// TIA Portal V16 export
// export: Created 2024-09-05T17:39:16.5674973Z, ExportSetting WithDefaults, DisplayName Totally Integrated Automation Portal, DisplayVersion V16 Update 6, DisplayName TIA Portal Version Control Interface, DisplayVersion V16 Update 2, DisplayName TIA Portal Openness, DisplayVersion V16 Update 6, DisplayName STEP 7 Professional, DisplayVersion V16 Update 6, DisplayName STEP 7 Safety, DisplayVersion V16, DisplayName WinCC Advanced, DisplayVersion V16 Update 6
DATA_BLOCK "DB_ProductionProgramEdit"   // DB6103
{ S7_Optimized_Access := 'FALSE' }
VERSION : 0.1
// stored: AutoNumber false, DBAccessibleFromOPCUA true, IsOnlyStoredInLoadMemory false, IsWriteProtectedInAS false
   VAR
      ProgramEmpty { S7_SetPoint := 'True'} : "UDT_ProductionProgram";
      ProgramInBox { S7_SetPoint := 'True'} : "UDT_ProductionProgram";
      ProgramEdit { S7_SetPoint := 'True'} : "UDT_ProductionProgram";
      Commands : Struct
         ProgramEdit : Struct
            Number : UInt := 5;
            NumberLast : UInt := 5;
            NumberChanged : Bool := FALSE;
            NumberInBox : UInt := 5;
            Commands : UInt := 0;   // 1= Load, 2= Save, 3= Copy, 4= Paste, 5= Delete
            LoadAll : Bool := FALSE;
            ProgramChanged : Bool := FALSE;
            SettingsCanBeChanged : Bool := TRUE;
            ChangeButtonsBlinking : Bool := FALSE;
            ChangeButtonsVisibility : Bool := FALSE;
            CommandsVisibility : Bool := TRUE;
         END_STRUCT;
         ProductEdit : Struct
            Number : UInt := 1;
            NumberLast : UInt := 1;
            NumberChanged : Bool := FALSE;
            Load : Bool := FALSE;
         END_STRUCT;
         PositionEdit : Struct
            Number : UInt := 1;
            NumberLast : UInt := 1;
            NumberChanged : Bool := FALSE;
            Load : Bool := FALSE;
         END_STRUCT;
      END_STRUCT;
   END_VAR
BEGIN
   ProgramEmpty."Name" := '';
   ProgramEmpty.CupformingParametersLeft.DigiforceProgram := 0;
   ProgramEmpty.CupformingParametersLeft.FinalSpeed := 0.0;
   ProgramEmpty.CupformingParametersLeft.ApproachSpeed := 0.0;
   ProgramEmpty.CupformingParametersLeft.FinalForce := 0.0;
   ProgramEmpty.CupformingParametersLeft.ApproachForce := 0.0;
   ProgramEmpty.CupformingParametersLeft.EndWayImmediate := 0.0;
   ProgramEmpty.CupformingParametersLeft.EndWayWithTimeout := 0.0;
   ProgramEmpty.CupformingParametersLeft.SwitchingWay := 0.0;
   ProgramEmpty.CupformingParametersLeft.EndWayTimeout := T#0MS;
   ProgramEmpty.CupformingParametersRight.DigiforceProgram := 0;
   ProgramEmpty.CupformingParametersRight.FinalSpeed := 0.0;
   ProgramEmpty.CupformingParametersRight.ApproachSpeed := 0.0;
   ProgramEmpty.CupformingParametersRight.FinalForce := 0.0;
   ProgramEmpty.CupformingParametersRight.ApproachForce := 0.0;
   ProgramEmpty.CupformingParametersRight.EndWayImmediate := 0.0;
   ProgramEmpty.CupformingParametersRight.EndWayWithTimeout := 0.0;
   ProgramEmpty.CupformingParametersRight.SwitchingWay := 0.0;
   ProgramEmpty.CupformingParametersRight.EndWayTimeout := T#0MS;
   ProgramEmpty.St1Insertion[1..20] := FALSE;
   ProgramEmpty.St1InsertionUsed[1..20] := FALSE;
   ProgramEmpty.FaureciaNumber := '';
   ProgramEmpty.FaureciaNumberStartChar := 0;
   ProgramEmpty.FaureciaNumberLength := 0;
   ProgramEmpty.MechanicalType := 0;
   ProgramInBox."Name" := 'startup';
   ProgramInBox.CupformingParametersLeft.DigiforceProgram := 1;
   ProgramInBox.CupformingParametersLeft.FinalSpeed := 25.0;
   ProgramInBox.CupformingParametersLeft.ApproachSpeed := 25.0;
   ProgramInBox.CupformingParametersLeft.FinalForce := 10.0;
   ProgramInBox.CupformingParametersLeft.ApproachForce := 10.0;
   ProgramInBox.CupformingParametersLeft.EndWayImmediate := 2.55;
   ProgramInBox.CupformingParametersLeft.EndWayWithTimeout := 3.0;
   ProgramInBox.CupformingParametersLeft.SwitchingWay := 20.0;
   ProgramInBox.CupformingParametersLeft.EndWayTimeout := T#300MS;
   ProgramInBox.CupformingParametersRight.DigiforceProgram := 1;
   ProgramInBox.CupformingParametersRight.FinalSpeed := 25.0;
   ProgramInBox.CupformingParametersRight.ApproachSpeed := 25.0;
   ProgramInBox.CupformingParametersRight.FinalForce := 60.0;
   ProgramInBox.CupformingParametersRight.ApproachForce := 10.0;
   ProgramInBox.CupformingParametersRight.EndWayImmediate := 2.7;
   ProgramInBox.CupformingParametersRight.EndWayWithTimeout := 3.0;
   ProgramInBox.CupformingParametersRight.SwitchingWay := 20.0;
   ProgramInBox.CupformingParametersRight.EndWayTimeout := T#300MS;
   ProgramInBox.St1Insertion[1] := TRUE;
   ProgramInBox.St1Insertion[2] := FALSE;
   ProgramInBox.St1Insertion[3..5] := TRUE;
   ProgramInBox.St1Insertion[6] := FALSE;
   ProgramInBox.St1Insertion[7] := TRUE;
   ProgramInBox.St1Insertion[8] := FALSE;
   ProgramInBox.St1Insertion[9..10] := TRUE;
   ProgramInBox.St1Insertion[11] := FALSE;
   ProgramInBox.St1Insertion[12..17] := TRUE;
   ProgramInBox.St1Insertion[18] := FALSE;
   ProgramInBox.St1Insertion[19] := TRUE;
   ProgramInBox.St1Insertion[20] := FALSE;
   ProgramInBox.St1InsertionUsed[1..7] := TRUE;
   ProgramInBox.St1InsertionUsed[8] := FALSE;
   ProgramInBox.St1InsertionUsed[9..19] := TRUE;
   ProgramInBox.St1InsertionUsed[20] := FALSE;
   ProgramInBox.FaureciaNumber := '2567208X';
   ProgramInBox.FaureciaNumberStartChar := 9;
   ProgramInBox.FaureciaNumberLength := 8;
   ProgramInBox.MechanicalType := 0;
   ProgramEdit."Name" := 'startup';
   ProgramEdit.CupformingParametersLeft.DigiforceProgram := 1;
   ProgramEdit.CupformingParametersLeft.FinalSpeed := 25.0;
   ProgramEdit.CupformingParametersLeft.ApproachSpeed := 25.0;
   ProgramEdit.CupformingParametersLeft.FinalForce := 10.0;
   ProgramEdit.CupformingParametersLeft.ApproachForce := 10.0;
   ProgramEdit.CupformingParametersLeft.EndWayImmediate := 2.55;
   ProgramEdit.CupformingParametersLeft.EndWayWithTimeout := 3.0;
   ProgramEdit.CupformingParametersLeft.SwitchingWay := 20.0;
   ProgramEdit.CupformingParametersLeft.EndWayTimeout := T#300MS;
   ProgramEdit.CupformingParametersRight.DigiforceProgram := 1;
   ProgramEdit.CupformingParametersRight.FinalSpeed := 25.0;
   ProgramEdit.CupformingParametersRight.ApproachSpeed := 25.0;
   ProgramEdit.CupformingParametersRight.FinalForce := 60.0;
   ProgramEdit.CupformingParametersRight.ApproachForce := 10.0;
   ProgramEdit.CupformingParametersRight.EndWayImmediate := 2.7;
   ProgramEdit.CupformingParametersRight.EndWayWithTimeout := 3.0;
   ProgramEdit.CupformingParametersRight.SwitchingWay := 20.0;
   ProgramEdit.CupformingParametersRight.EndWayTimeout := T#300MS;
   ProgramEdit.St1Insertion[1] := TRUE;
   ProgramEdit.St1Insertion[2] := FALSE;
   ProgramEdit.St1Insertion[3..5] := TRUE;
   ProgramEdit.St1Insertion[6] := FALSE;
   ProgramEdit.St1Insertion[7] := TRUE;
   ProgramEdit.St1Insertion[8] := FALSE;
   ProgramEdit.St1Insertion[9..10] := TRUE;
   ProgramEdit.St1Insertion[11] := FALSE;
   ProgramEdit.St1Insertion[12..17] := TRUE;
   ProgramEdit.St1Insertion[18] := FALSE;
   ProgramEdit.St1Insertion[19] := TRUE;
   ProgramEdit.St1Insertion[20] := FALSE;
   ProgramEdit.St1InsertionUsed[1..7] := TRUE;
   ProgramEdit.St1InsertionUsed[8] := FALSE;
   ProgramEdit.St1InsertionUsed[9..19] := TRUE;
   ProgramEdit.St1InsertionUsed[20] := FALSE;
   ProgramEdit.FaureciaNumber := '2567208X';
   ProgramEdit.FaureciaNumberStartChar := 9;
   ProgramEdit.FaureciaNumberLength := 8;
   ProgramEdit.MechanicalType := 0;
END_DATA_BLOCK
